// TIA Portal V17 export
// export: Created 2024-09-03T21:55:01.3642666Z, ExportSetting WithDefaults, DisplayName Totally Integrated Automation Portal, DisplayVersion V17 Update 7, DisplayName TIA Portal Openness, DisplayVersion V17 Update 7, DisplayName TIA Portal Version Control Interface, DisplayVersion V17, DisplayName SINAMICS Startdrive Advanced, DisplayVersion V17 SP2, DisplayName SINAMICS Startdrive G110M, G120, G120C, G120D, G120P, G115D, DisplayVersion V17 SP2, DisplayName SINAMICS Startdrive G130, G150, S120, S150, SINAMICS MV, S210, DisplayVersion V17 SP2, DisplayName STEP 7 Professional, DisplayVersion V17 Update 7, DisplayName STEP 7 Safety, DisplayVersion V17 Update 6, DisplayName WinCC Advanced / Unified PC, DisplayVersion V17 Update 7
FUNCTION_BLOCK "FB_IJC"   // FB800, LAD
{ S7_Optimized_Access := 'TRUE' }
VERSION : 0.1
// stored: AutoNumber false, IsIECCheckEnabled false, IsRetainMemResEnabled false, MemoryReserve 100, SetENOAutomatically false, UDAEnableTagReadback false
   VAR
      MSG { S7_SetPoint := 'True'} : Array[0..30] of "IJC PROTOCOL";
      NFP_1 { S7_SetPoint := 'True'} : String[8];
      Component_1 : String[30];
      NFP_2 : String[8];
      Component_2 : String[30];
      Send_STA : Array[0..5] of Bool;
      Send_TRC : Array[0..5] of Bool;
      Send_TRR : Array[0..5] of Bool;
      Send_CNF : Array[0..5] of Bool;
      IJC_STA_1_Ans_OK : Bool;
      IJC_STA_1_Ans_NOK : Bool;
      IJC_TRC_1_Ans_OK : Bool;
      IJC_TRC_1_Ans_NOK : Bool;
      IJC_STA_2_Ans_NOK : Bool;
      IJC_STA_2_Ans_OK : Bool;
      IJC_TRC_2_Ans_OK : Bool;
      IJC_TRC_2_Ans_NOK : Bool;
      FP1 : Bool;
      FP2 : Bool;
      FP3 : Bool;
      FP4 : Bool;
      FP5 : Bool;
      FP6 : Bool;
      Reset : Bool;
      IJC_Enable : Bool;
      DN_STA : Array[0..5] of Bool;
      DN_TRC : Array[0..5] of Bool;
      DN_TRR : Array[0..5] of Bool;
      DN_CNF : Array[0..5] of Bool;
      INDEX : Int;
      ALL_STA_OK : Bool;
      AWAKE_SIGNAL_INSTANCE : "AWAKE_SIGNAL";
   END_VAR
   VAR_TEMP
      i : USInt;
      res : SInt;
      INDEX_NFP : Int;
   END_VAR
BEGIN

REGION Network 1
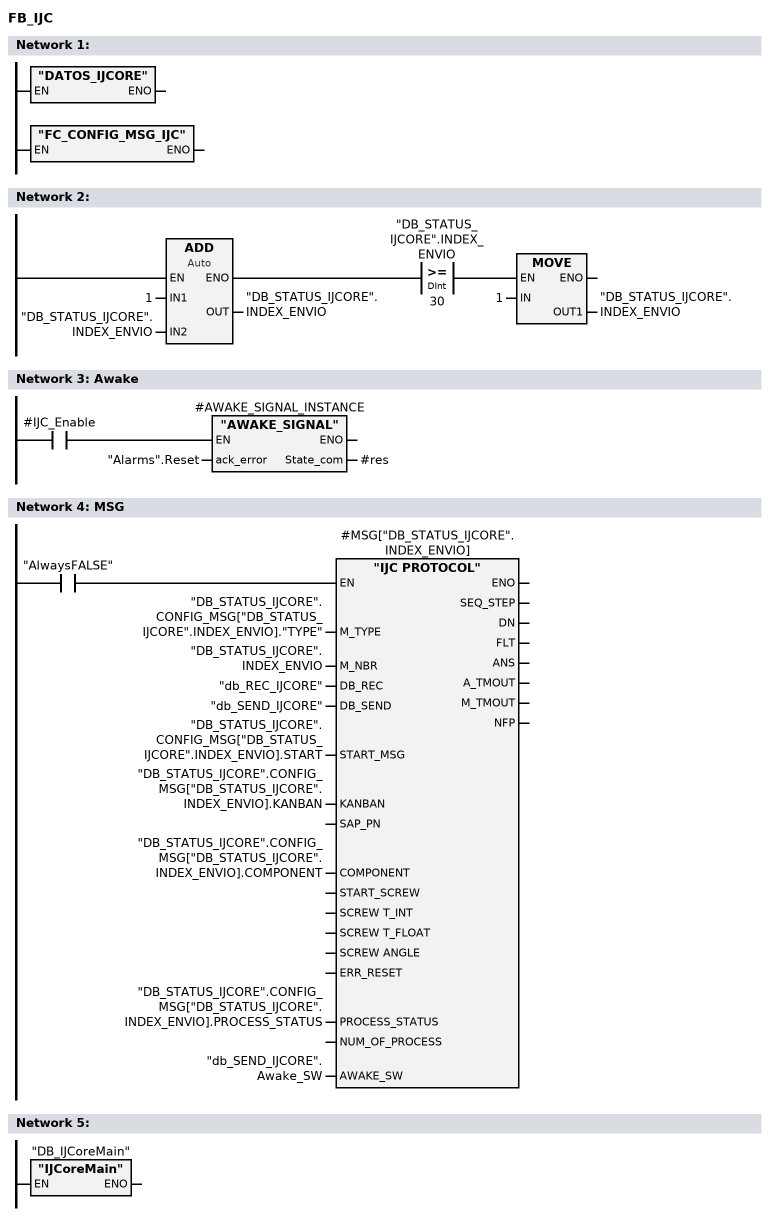
   RUNG wire#powerrail
      "DATOS_IJCORE"()
   END_RUNG
   RUNG wire#powerrail
      "FC_CONFIG_MSG_IJC"()
   END_RUNG
   // the same network as SCL:
   "DATOS_IJCORE"();
   "FC_CONFIG_MSG_IJC"();
END_REGION

REGION Network 2
   RUNG wire#powerrail
      Add(in1 := 1, in2 := "DB_STATUS_IJCORE".INDEX_ENVIO, out => "DB_STATUS_IJCORE".INDEX_ENVIO)
      { S7_Templates := "SrcType := DInt" } GE_Contact(in1 := "DB_STATUS_IJCORE".INDEX_ENVIO, in2 := 30)
      Move(in := 1, out1 => "DB_STATUS_IJCORE".INDEX_ENVIO)
   END_RUNG
   // the same network as SCL:
   "DB_STATUS_IJCORE".INDEX_ENVIO := 1 + "DB_STATUS_IJCORE".INDEX_ENVIO;
   IF "DB_STATUS_IJCORE".INDEX_ENVIO >= 30 THEN "DB_STATUS_IJCORE".INDEX_ENVIO := 1; END_IF;
END_REGION

REGION Network 3: Awake
   RUNG wire#powerrail
      Contact( #IJC_Enable )
      #AWAKE_SIGNAL_INSTANCE(ack_error := "Alarms".Reset, State_com => #res)
   END_RUNG
   // the same network as SCL:
   IF #IJC_Enable THEN
       #AWAKE_SIGNAL_INSTANCE(ack_error := "Alarms".Reset, State_com => #res);   // "AWAKE_SIGNAL"
   END_IF;
END_REGION

REGION Network 4: MSG
   RUNG wire#powerrail
      Contact( "AlwaysFALSE" )
      #MSG["DB_STATUS_IJCORE".INDEX_ENVIO](M_TYPE := "DB_STATUS_IJCORE".CONFIG_MSG["DB_STATUS_IJCORE".INDEX_ENVIO]."TYPE", M_NBR := "DB_STATUS_IJCORE".INDEX_ENVIO, DB_REC := "db_REC_IJCORE", DB_SEND := "db_SEND_IJCORE", START_MSG := "DB_STATUS_IJCORE".CONFIG_MSG["DB_STATUS_IJCORE".INDEX_ENVIO].START, KANBAN := "DB_STATUS_IJCORE".CONFIG_MSG["DB_STATUS_IJCORE".INDEX_ENVIO].KANBAN, SAP_PN :=, COMPONENT := "DB_STATUS_IJCORE".CONFIG_MSG["DB_STATUS_IJCORE".INDEX_ENVIO].COMPONENT, START_SCREW :=, "SCREW T_INT" :=, "SCREW T_FLOAT" :=, "SCREW ANGLE" :=, ERR_RESET :=, PROCESS_STATUS := "DB_STATUS_IJCORE".CONFIG_MSG["DB_STATUS_IJCORE".INDEX_ENVIO].PROCESS_STATUS, NUM_OF_PROCESS :=, AWAKE_SW := "db_SEND_IJCORE".Awake_SW, SEQ_STEP =>, DN =>, FLT =>, ANS =>, A_TMOUT =>, M_TMOUT =>, NFP =>)
   END_RUNG
   // the same network as SCL:
   IF "AlwaysFALSE" THEN
       #MSG["DB_STATUS_IJCORE".INDEX_ENVIO](M_TYPE := "DB_STATUS_IJCORE".CONFIG_MSG["DB_STATUS_IJCORE".INDEX_ENVIO]."TYPE",   // "IJC PROTOCOL"
                               M_NBR := "DB_STATUS_IJCORE".INDEX_ENVIO,
                               DB_REC := "db_REC_IJCORE",
                               DB_SEND := "db_SEND_IJCORE",
                               START_MSG := "DB_STATUS_IJCORE".CONFIG_MSG["DB_STATUS_IJCORE".INDEX_ENVIO].START,
                               KANBAN := "DB_STATUS_IJCORE".CONFIG_MSG["DB_STATUS_IJCORE".INDEX_ENVIO].KANBAN,
                               COMPONENT := "DB_STATUS_IJCORE".CONFIG_MSG["DB_STATUS_IJCORE".INDEX_ENVIO].COMPONENT,
                               PROCESS_STATUS := "DB_STATUS_IJCORE".CONFIG_MSG["DB_STATUS_IJCORE".INDEX_ENVIO].PROCESS_STATUS,
                               AWAKE_SW := "db_SEND_IJCORE".Awake_SW);
   END_IF;
END_REGION

REGION Network 5
   RUNG wire#powerrail
      "DB_IJCoreMain"()
   END_RUNG
   // the same network as SCL:
   "DB_IJCoreMain"();   // "IJCoreMain"
END_REGION
END_FUNCTION_BLOCK
